// TwinCAT 3 PLC project Library
// Title: lcls-twincat-motion
// Company: SLAC
// ProjectVersion: 0.0.0
// ProgramVersion: 3.1.4020.5
// libraries:
//   LCLS General, * (SLAC)
//   PMPS, * (SLAC - LCLS)
//   Tc2_EtherCAT, * (Beckhoff Automation GmbH)
//   Tc2_MC2, * (Beckhoff Automation GmbH)
//   Tc2_Standard, * (Beckhoff Automation GmbH)
//   Tc2_System, * (Beckhoff Automation GmbH)
//   Tc2_Utilities, * (Beckhoff Automation GmbH)
//   Tc3_JsonXml, * (Beckhoff Automation GmbH)
//   Tc3_Module, * (Beckhoff Automation GmbH)
// project tree:
//   DUTs/ DUT_MotionStage.TcDUT, DUT_MotionStageNCParams.TcDUT, DUT_PositionState.TcDUT (not stored), EL5042_Status.TcDUT (not stored), ENUM_EpicsHomeCmd.TcDUT (not stored), ENUM_EpicsInOut.TcDUT (not stored), ENUM_EpicsMotorCmd.TcDUT (not stored), ENUM_MotionRequest.TcDUT (not stored), ENUM_StageBrakeMode.TcDUT (not stored), ENUM_StageEnableMode.TcDUT (not stored), DUT_MotionPneumaticActuator.TcDUT (not stored), ENUM_PnuematicActuatorPositionState.TcDUT (not stored), ST_RenishawAbsEnc.TcDUT (not stored)
//   GVLs/ MOTION_GVL.TcGVL (not stored)
//   / PlcTask.TcTTO (not stored)
//   POUs/Deprecated/ FB_EpicsInOut.TcPOU (not stored), FB_PositionStateManager.TcPOU (not stored), FB_StatePTPMove.TcPOU (not stored)
//   POUs/ImplicitChecks/ CheckBounds.TcPOU (not stored), CheckDivDInt.TcPOU (not stored), CheckDivLInt.TcPOU (not stored), CheckDivLReal.TcPOU (not stored), CheckDivReal.TcPOU (not stored)
//   POUs/Motion/ FB_EncoderValue.TcPOU (not stored), FB_EncSaveRestore.TcPOU (not stored), FB_LogMotionError.TcPOU (not stored), FB_MotionHoming.TcPOU (not stored), FB_MotionRequest.TcPOU (not stored), FB_MotionStage.TcPOU (not stored), FB_MotionStageNCParams.TcPOU, FB_MotionStageSim.TcPOU (not stored), FB_MotionPneumaticActuator.TcPOU (not stored)
//   POUs/Motion/Gantry/ FB_GantryAutoCoupling.TcPOU (not stored), FB_GantryDiffVirtualLimitSwitch.TcPOU (not stored)
//   POUs/Motion/PMPS/ FB_EncErrorFFO.TcPOU (not stored), FB_PositionStatePMPS.TcPOU (not stored), FB_NCErrorFFO.TcPOU (not stored), FB_PositionStatePMPS_Base.TcPOU (not stored), FB_PositionStatePMPS_Test.TcPOU (not stored)
//   POUs/Motion/States/Examples/ FB_PositionStateInOut.TcPOU (not stored), FB_PositionStateInOut_WithPMPS.TcPOU (not stored), FB_PositionStateInOut_WithPMPS_Test.TcPOU (not stored)
//   POUs/Motion/States/ FB_PositionStateBase.TcPOU (not stored), FB_PositionStateBase_WithPMPS.TcPOU (not stored), FB_PositionStateBase_WithPMPS_Test.TcPOU (not stored), FB_PositionStateMove.TcPOU (not stored)
//   POUs/Motion/States/Helpers/ FB_RawCountConverter.TcPOU (not stored), F_AtPositionState.TcPOU (not stored), F_PosOverLowerBound.TcPOU (not stored), F_PosUnderUpperBound.TcPOU (not stored), F_PosWithinDelta.TcPOU (not stored)
//   POUs/Motion/States/Internals/ FB_PositionStateInternal.TcPOU (not stored), FB_PositionStateLock.TcPOU (not stored)
//   POUs/Motion/Utils/ FB_SetEnables.TcPOU (not stored), F_MotionErrorCodeLookup.TcPOU (not stored)
//   POUs/MotorTesting/ FB_MicroStepCountTest.TcPOU (not stored)
//   tc_mca_std_lib/DUTs/ DUT_AxisStatus_v0_01.TcDUT (not stored)
//   tc_mca_std_lib/GVLs/ GVL.TcGVL (not stored)
//   tc_mca_std_lib/POUs/ChangeConfig/ FB_ReadFloatParameter.TcPOU (not stored), FB_ReadParameterInNc_v1_00.TcPOU (not stored), FB_WriteFloatParameter.TcPOU (not stored), FB_WriteParameterInNc_v1_00.TcPOU (not stored)
//   tc_mca_std_lib/POUs/ErrorHandling/ DUT_ErrorState.TcDUT (not stored), DUT_TerminalError.TcDUT (not stored), FB_ErrorList.TcPOU (not stored), FB_TerminalError.TcPOU (not stored), GVL_ErrorSystem.TcGVL (not stored), ST_ErrorSystem.TcDUT (not stored)
//   tc_mca_std_lib/POUs/Hardware/EtherCAT_Terminals/Analog_Inputs/ EL3174_0002.TcPOU (not stored), EL3214.TcPOU (not stored), EL3255.TcPOU (not stored), FB_CalculateFrequency_3702_v0_01.TcPOU (not stored)
//   tc_mca_std_lib/POUs/Hardware/EtherCAT_Terminals/Digital_Inputs/ EL1008.TcPOU (not stored), EL1018.TcPOU (not stored), EL1808.TcPOU (not stored), EL1809.TcPOU (not stored), EL1819.TcPOU (not stored), FB_EL1252ASM_v1_00.TcPOU (not stored)
//   tc_mca_std_lib/POUs/Hardware/EtherCAT_Terminals/Digital_Outputs/ EL2014.TcPOU (not stored), EL2252.TcPOU (not stored), EL2808.TcPOU (not stored), EL2819.TcPOU (not stored)
//   tc_mca_std_lib/POUs/Hardware/EtherCAT_Terminals/Digital_Outputs/External_Types/ dutEL2521_Ctrl.TcDUT (not stored), dutEL2521_Status.TcDUT (not stored)
//   tc_mca_std_lib/POUs/Hardware/EtherCAT_Terminals/Measuring_Terminals/ EL5002.TcPOU (not stored), EL5021.TcPOU (not stored), EL5042.TcPOU (not stored), EL5101.TcPOU (not stored)
//   tc_mca_std_lib/POUs/Hardware/EtherCAT_Terminals/Motion/ EL7211_v1_00.TcPOU (not stored), EL9576_v1_00.TcPOU (not stored)
//   tc_mca_std_lib/POUs/Hardware/EtherCAT_Terminals/System/ EL9410.TcPOU (not stored), EL9505.TcPOU (not stored)
//   tc_mca_std_lib/POUs/Hardware/Other/ EK1200.TcPOU (not stored)
//   tc_mca_std_lib/POUs/Motion/ FB_DriveVirtual.TcPOU (not stored), FB_NcAxis.TcPOU (not stored)
//   tc_mca_std_lib/POUs/Motion/Homing/ FB_HomeDirect.TcPOU (not stored), FB_HomeFinish.TcPOU (not stored), FB_HomePrepare.TcPOU (not stored), FB_HomeReadNcVelocities.TcPOU (not stored), FB_HomeReadSoftLimEnable.TcPOU (not stored), FB_HomeToSwitch.TcPOU (not stored), FB_HomeVirtual.TcPOU (not stored), FB_HomeWriteNcVelocities.TcPOU (not stored), FB_HomeWriteSoftLimEnable.TcPOU (not stored)
//   UnitTests/ BasicTests.TcPOU (not stored), Interactive.TcPOU (not stored)
//   Version/ Global_Version.TcGVL (not stored)

// ---- DUTs/DUT_MotionStage.TcDUT
TYPE DUT_MotionStage :
    // Defines the EPICS interface to moving a motor in TwinCAT
STRUCT
(* Hardware *)

    // PLC Axis Reference
    Axis: AXIS_REF;
    // NC Forward Limit Switch: TRUE if ok to move
    {attribute 'pytmc' := '
        pv: PLC:bLimitForwardEnable
        io: i
        field: ZNAM FALSE
        field: ONAM TRUE
        field: DESC FALSE if forward limit hit
    '}
    bLimitForwardEnable AT %I*: BOOL;
    // NC Backward Limit Switch: TRUE if ok to move
    {attribute 'pytmc' := '
        pv: PLC:bLimitBackwardEnable
        io: i
        field: ZNAM FALSE
        field: ONAM TRUE
        field: DESC FALSE if reverse limit hit
    '}
    bLimitBackwardEnable AT %I*: BOOL;
    // NO Home Switch: TRUE if at home
    {attribute 'pytmc' := '
        pv: PLC:bHome
        io: i
        field: ZNAM FALSE
        field: ONAM TRUE
        field: DESC TRUE if at homing switch
    '}
    bHome AT %I*: BOOL;
    // NC Brake Output: TRUE to release brake
    {attribute 'pytmc' := '
        pv: PLC:bBrakeRelease
        io: i
        field: ZNAM FALSE
        field: ONAM TRUE
        field: DESC TRUE if brake released
    '}
    bBrakeRelease AT %Q*: BOOL;
    // NC STO Input: TRUE if ok to move
    {attribute 'pytmc' := '
        pv: PLC:bHardwareEnable
        io: i
        field: ZNAM FALSE
        field: ONAM TRUE
        field: DESC TRUE if STO not hit
    '}
    bHardwareEnable AT %I*: BOOL;

    // Raw encoder IO for ULINT (Biss-C)
    nRawEncoderULINT AT %I*: ULINT;
    // Raw encoder IO for UINT (Relative Encoders)
    nRawEncoderUINT AT %I*: UINT;
    // Raw encoder IO for INT (LVDT)
    nRawEncoderINT AT %I*: INT;

    (* Psuedo-hardware *)

    // Forward enable EPS summary
    {attribute 'pytmc' := '
        pv: PLC:bAllForwardEnable
        io: i
        field: ZNAM FALSE
        field: ONAM TRUE
        field: DESC Summary of axis permission to move forward
    '}
    bAllForwardEnable: BOOL:=FALSE;
    // Backward enable EPS summary
    {attribute 'pytmc' := '
        pv: PLC:bAllBackwardEnable
        io: i
        field: ZNAM FALSE
        field: ONAM TRUE
        field: DESC Summary of axis permission to move backward
    '}
    bAllBackwardEnable: BOOL:=FALSE;
    // Enable EPS summary encapsulating emergency stop button and any additional motion preventive hardware
    {attribute 'pytmc' := '
        pv: PLC:bAllEnable
        io: i
        field: ZNAM FALSE
        field: ONAM TRUE
        field: DESC Summary of axis permission to have power
    '}
    bAllEnable: BOOL:=FALSE;
    // Forward virtual gantry limit switch
    {attribute 'pytmc' := '
        pv: PLC:bGantryForwardEnable
        io: i
        field: ZNAM FALSE
        field: ONAM TRUE
        field: DESC TRUE if gantry ok to move forward
    '}
    bGantryForwardEnable: BOOL:=FALSE;
    // Backward virtual gantry limit switch
    {attribute 'pytmc' := '
        pv: PLC:bGantryBackwardEnable
        io: i
        field: ZNAM FALSE
        field: ONAM TRUE
        field: DESC TRUE if gantry ok to move backward
    '}
    bGantryBackwardEnable: BOOL:=FALSE;
    // Encoder count summary, if linked above
    {attribute 'pytmc' := '
        pv: PLC:nEncoderCount
        io: i
        field: DESC Count from encoder hardware
    '}
    nEncoderCount: UDINT;

    (* Settings *)
    // Name to use for log messages, fast faults, etc.
    {attribute 'pytmc' := '
        pv: PLC:sName
        io: i
        field: DESC PLC program name
    '}
    sName: STRING;
    // If TRUE, we want to enable the motor independently of PMPS or other safety systems.
    {attribute 'pytmc' := '
        pv: PLC:bPowerSelf
        io: i
        field: ZNAM FALSE
        field: ONAM TRUE
        field: DESC FALSE if axis is in PMPS
    '}
    bPowerSelf: BOOL:=FALSE;
    // Determines when we automatically enable the motor
    {attribute 'pytmc' := '
        pv: PLC:nEnableMode
        io: i
        field: DESC Describes when the axis will automatically get power
    '}
    nEnableMode: ENUM_StageEnableMode:=ENUM_StageEnableMode.DURING_MOTION;
    // Determines when we automatically disengage the brake
    {attribute 'pytmc' := '
        pv: PLC:nBrakeMode
        io: i
        field: DESC Describes when the brake will be released
    '}
    nBrakeMode: ENUM_StageBrakeMode:=ENUM_StageBrakeMode.IF_ENABLED;
    // Determines our encoder homing strategy
    {attribute 'pytmc' := '
        pv: PLC:nHomingMode
        io: i
        field: DESC Describes our homing strategy
    '}
    nHomingMode: ENUM_EpicsHomeCmd:=ENUM_EpicsHomeCmd.NONE;
    // Set true to activate gantry EPS
    {attribute 'pytmc' := '
        pv: PLC:bGantryAxis
        io: i
        field: ZNAM FALSE
        field: ONAM TRUE
        field: DESC TRUE if gantry EPS active
    '}
    bGantryAxis: BOOL:=FALSE;

    // Set to gantry difference tolerance
    nGantryTol: LINT:=0;

    // Encoder count at which this axis is aligned with other axis
    nEncRef: ULINT:=0;

    (* Commands *)
    // Used internally to request enables
    {attribute 'pytmc' := '
        pv: PLC:bEnable
        io: io
        field: ZNAM FALSE
        field: ONAM TRUE
        field: DESC Used internally to request enables
    '}
    bEnable: BOOL;
    // Used internally to reset errors and other state
    {attribute 'pytmc' := '
        pv: PLC:bReset
        io: io
        field: ZNAM FALSE
        field: ONAM TRUE
        field: DESC Used internally to reset errors
    '}
    bReset: BOOL;
    // Used internally and by the IOC to start or stop a move
    {attribute 'pytmc' := '
        pv: PLC:bExecute
        io: io
        field: ZNAM FALSE
        field: ONAM TRUE
        field: DESC Used internally and by the IOC to start or stop
    '}
    bExecute: BOOL;
    // Used by the IOC to disable an axis
    {attribute 'pytmc' := '
        pv: PLC:bUserEnable
        io: io
        field: ZNAM DISABLE
        field: ONAM ENABLE
        field: DESC Used to disable power entirely for an axis
    '}
    bUserEnable: BOOL := 1;

    (* Shortcut Commands *)
    // Start a move to fPosition with fVelocity
    {attribute 'pytmc' := '
        pv: PLC:bMoveCmd
        io: io
        field: DESC Start a move
    '}
    bMoveCmd: BOOL;
    // Start the homing routine
    {attribute 'pytmc' := '
        pv: PLC:bHomeCmd
        io: io
        field: DESC Start the homing routine
    '}
    bHomeCmd: BOOL;

    (* Command Args *)
    // Used internally and by the IOC to pick what kind of move to do
    {attribute 'pytmc' := '
        pv: PLC:nCommand
        io: io
        field: DESC Used internally and by the IOC to pick move type
    '}
    nCommand: INT;
    // Used internally and by the IOC to pass additional data to some commands
    {attribute 'pytmc' := '
        pv: PLC:nCmdData
        io: io
        field: DESC Used internally and by the IOC to pass extra args
    '}
    nCmdData: INT;
    // Used internally and by the IOC to pick a destination for the move
    {attribute 'pytmc' := '
        pv: PLC:fPosition
        io: io
        field: DESC Used internally and by the IOC as the set position
    '}
    fPosition: LREAL;
    // Used internally and by the IOC to pick a move velocity
    {attribute 'pytmc' := '
        pv: PLC:fVelocity
        io: io
        field: DESC Used internally and by the IOC to set velocity
    '}
    fVelocity: LREAL;
    // Used internally and by the IOC to pick a move acceleration
    {attribute 'pytmc' := '
        pv: PLC:fAcceleration
        io: io
        field: DESC Used internally and by the IOC to set acceleration
    '}
    fAcceleration: LREAL;
    // Used internally and by the IOC to pick a move deceleration
    {attribute 'pytmc' := '
        pv: PLC:fDeceleration
        io: io
        field: DESC Used internally and by the IOC to set deceleration
    '}
    fDeceleration: LREAL;
    // Used internally and by the IOC to pick a home position
    {attribute 'pytmc' := '
        pv: PLC:fHomePosition
        io: io
        field: DESC Used internally and by the IOC to pick home position
    '}
    fHomePosition: LREAL;

    (* Info *)
    // Unique ID assigned to each axis in the NC
    {attribute 'pytmc' := '
        pv: PLC:nMotionAxisID
        io: i
        field: DESC Unique ID assigned to each axis in the NC
    '}
    nMotionAxisID: UDINT:=0;

    (* Returns *)
    // TRUE if done enabling
    {attribute 'pytmc' := '
        pv: PLC:bEnableDone
        io: i
        field: ZNAM FALSE
        field: ONAM TRUE
        field: DESC TRUE if done enabling
    '}
    bEnableDone: BOOL;
    // TRUE if in the middle of a command
    {attribute 'pytmc' := '
        pv: PLC:bBusy
        io: i
        field: ZNAM FALSE
        field: ONAM TRUE
        field: DESC TRUE if in the middle of a command
    '}
    bBusy: BOOL;
    // TRUE if we've done a command and it has finished
    {attribute 'pytmc' := '
        pv: PLC:bDone
        io: i
        field: ZNAM FALSE
        field: ONAM TRUE
        field: DESC TRUE if command finished successfully
    '}
    bDone: BOOL;
    // TRUE if the motor has been homed, or does not need to be homed
    {attribute 'pytmc' := '
        pv: PLC:bHomed
        io: i
        field: DESC TRUE if the motor has been homed
    '}
    bHomed: BOOL;
    // TRUE if we have safety permission to move
    {attribute 'pytmc' := '
        pv: PLC:bSafetyReady
        io: i
        field: ZNAM FALSE
        field: ONAM TRUE
        field: DESC TRUE if safe to start a move
    '}
    bSafetyReady: BOOL;
    // TRUE if we're in an error state
    {attribute 'pytmc' := '
        pv: PLC:bError
        io: i
        field: ZNAM FALSE
        field: ONAM TRUE
        field: DESC TRUE if we are in an error state
        update: 100Hz notify
    '}
    bError: BOOL;
    // Error code if nonzero
    {attribute 'pytmc' := '
        pv: PLC:nErrorId
        io: i
        field: DESC Error code if nonzero
        update: 100Hz notify
    '}
    nErrorId: UDINT;
    // Message to identify the error state
    {attribute 'pytmc' := '
        pv: PLC:sErrorMessage
        io: i
        field: DESC Message to identify the error state
        update: 100Hz notify
    '}
    sErrorMessage: STRING;
    // Internal hook for custom error messages
    sCustomErrorMessage: STRING;
    // MC_ReadParameterSet Output
    stAxisParameters: ST_AxisParameterSet;
    // True if we've updated stAxisParameters at least once
    bAxisParamsInit: BOOL;

    // Misc axis status information for the IOC
    stAxisStatus: DUT_AxisStatus_v0_01;

    (* Other status information for users of the IOC *)
    // Position lag difference
    {attribute 'pytmc' := '
        pv: PLC:fPosDiff
        io: i
        field: DESC Position lag difference
    '}
    fPosDiff: LREAL;
    //create parameters for struct of published PV's
    {attribute 'pytmc' := '
        pv: NC
        io: i
        field: DESC Position lag difference
    '}
    stMotionStageNCParams: DUT_MotionStageNCParams;
END_STRUCT
END_TYPE

// ---- DUTs/DUT_MotionStageNCParams.TcDUT
TYPE DUT_MotionStageNCParams :
STRUCT
    // NC Forward Limit Switch: TRUE if ok to move
    {attribute 'pytmc' := '
        pv: FEncOffset
        io: i
        field: ZNAM FALSE
        field: ONAM TRUE
        field: DESC FALSE if forward limit hit
    '}
    fEncOffset AT %I*: LREAL;
    // NC Backward Limit Switch: TRUE if ok to move
    {attribute 'pytmc' := '
        pv: fEncScaleFactor
        io: i
        field: ZNAM FALSE
        field: ONAM TRUE
        field: DESC FALSE if reverse limit hit
    '}
    fEncScaleFactor AT %I*: LREAL;
    //test
END_STRUCT
END_TYPE

// ---- POUs/Motion/FB_MotionStageNCParams.TcPOU
FUNCTION_BLOCK FB_MotionStageNCParams
(*
    Read and refresh axis parameters struct on DUT_MotionStage
*)
VAR_IN_OUT
    stMotionStage: DUT_MotionStage;
END_VAR
VAR_INPUT
    bEnable: BOOL;
    tRefreshDelay: TIME;
END_VAR
VAR_OUTPUT
    bError: BOOL;
END_VAR
VAR
    mcReadParams: MC_ReadParameterSet;
    timer: TON;
    bExecute: BOOL := TRUE;
    nLatchErrId: UDINT;
END_VAR

timer(
    IN:=bEnable AND NOT bExecute,
    PT:=tRefreshDelay);
bExecute S= timer.Q;
mcReadParams(
    Parameter:=stMotionStage.stAxisParameters,
    Axis:=stMotionStage.Axis,
    Execute:=bEnable AND bExecute,
    Error=>bError);
IF mcReadParams.ErrorID <> 0 THEN
    nLatchErrId := 0;
END_IF
bExecute R= mcReadParams.Done OR mcReadParams.Error;
stMotionStage.bAxisParamsInit S= mcReadParams.Done;
stMotionStage.stMotionStageNCParams.fEncOffset := stMotionStage.stAxisParameters.fEncOffset;
stMotionStage.stMotionStageNCParams.fEncScaleFactor := stMotionStage.stAxisParameters.fEncScaleFactorInternal;

END_FUNCTION_BLOCK
